# EPICS substitutions: IVU18App/Db/ivu18_motorstatus.substitutions
file "db/ivu18_motorstatus.template"
{
pattern
{AXIS, AXISNAME}
{"1", "GU"}
{"2", "GD"}
{"3", "EU"}
{"4", "ED"}
}
